# EPICS substitutions: iocBoot/iocnamWin/substitutions/fb_epid.substitutions
# $Id$

file "$(OPTICS)/opticsApp/Db/fb_epid.db"
  {
    {
        P=namWin:epid1,
	IN=namWin:epid1:sim.VAL,
	OUT=namWin:epid1:sim.D,
	MODE=PID,
	CALC=A,
	PERMIT1="namWin:epid1:on.VAL",
	PERMIT2="",
	PERMIT3="",
	PERMIT4=""
    }
  }
